/// TrackingMaster - Allows access to WindowTracking
INTERFACE I_TrackingMaster EXTENDS __SYSTEM.IQueryInterface

/// Tracking is ready for interactions (e.g. Conveyor is on constant speed)
PROPERTY P_TrackingReady : BOOL
GET
END_GET
END_PROPERTY

PROPERTY P_WindowTracking : I_WindowTracking
GET
END_GET
END_PROPERTY

END_INTERFACE

(* stored: Version 1.1.0.1, ProductVersion 3.1.4020.6
   Itf I_TrackingMaster: Id {2395bae8-fdae-4cdd-8797-46bb2496215e}
   Property P_TrackingReady: Id {aae3e85c-4b48-4f50-b5ce-86fec8576f0d}
   Get Get: Id {875e4818-6aa6-4dda-8935-53019a9cd610}
   Property P_WindowTracking: Id {c5787c80-d57e-4455-ac32-2f3848de25f5}
   Get Get: Id {8b2ab2bd-690b-4bea-8728-86546e45b9c3} *)
